PROGRAM MAIN
VAR
END_VAR

END_PROGRAM

(* stored: Version 1.1.0.1, ProductVersion 3.1.4024.14
   POU MAIN: Id {e0796ff0-ec64-4148-90f5-f2417ab607f2}, SpecialFunc None *)
